SUBAPPLICATION Uebung_008_AE (* Blinker mit E_CYCLE, E_SWITCH und E_SR *)
  (* Standard: 61499-2; Description: Copyright (c) 2023 Meisterschulen am Ostbahnhof This program and the accompanying materials are made available under the terms of the Eclipse Public License 2.0 which is available at https://www.eclipse.org/legal/epl-2.0/ SPDX-License-Identifier: EPL-2.0 *)
  (* Version 1.0, 2026-01-14, Franz Höpfinger, Meisterschulen am Ostbahnhof, initial API and implementation and/or initial documentation *)
  PACKAGE Uebungen;
  IMPORT logiBUS::io::DQ::logiBUS_DO::Output_Q1;
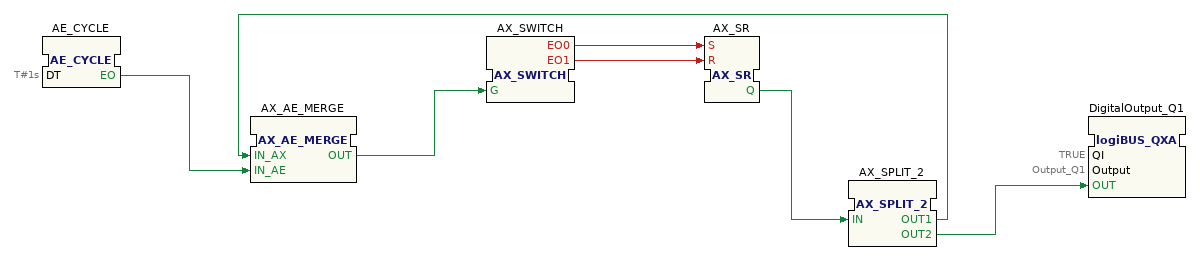
  FBS
    DigitalOutput_Q1 : logiBUS::io::DQ::logiBUS_QXA(QI := TRUE, Output := Output_Q1);
    AE_CYCLE : adapter::events::unidirectional::timers::AE_CYCLE(DT := T#1s);
    AX_SWITCH : adapter::events::unidirectional::AX_SWITCH;
    AX_SR : adapter::events::unidirectional::AX_SR;
    AX_SPLIT_2 : adapter::events::unidirectional::AX_SPLIT_2;
    AX_AE_MERGE : adapter::events::unidirectional::AX_AE_MERGE;
  END_FBS
  EVENT_CONNECTIONS
    AX_SWITCH.EO0 TO AX_SR.S;
    AX_SWITCH.EO1 TO AX_SR.R;
  END_CONNECTIONS
  ADAPTER_CONNECTIONS
    AX_SR.Q TO AX_SPLIT_2.IN;
    AX_SPLIT_2.OUT1 TO AX_AE_MERGE.IN_AX;
    AE_CYCLE.EO TO AX_AE_MERGE.IN_AE;
    AX_AE_MERGE.OUT TO AX_SWITCH.G;
    AX_SPLIT_2.OUT2 TO DigitalOutput_Q1.OUT;
  END_CONNECTIONS
END_SUBAPPLICATION
